(*
    private sync block removes the needs for circular interfaces variable passing amongs dependant Fbs
    that would otherwise lessen readability and complicate code scability and maintianing
    This block adds needed encapsulation for passing private data in write mode.
    it create a a communication buffer amongs synched function blocks; can also hold shareable feature implementation
    thus limititing the needs for addtional interface instantiation.
*)
{attribute 'hide_all_locals'}
FUNCTION_BLOCK FB_MotionSyncPrivate
VAR_INPUT
END_VAR
VAR_OUTPUT
END_VAR
VAR
    // private vars for data exchange
    eSyncPrvAxisState : MC_AxisStates;
    bSyncPrvReset : BOOL;
    bSyncPrvEnable :BOOL;
    bSyncPrvPowerEn : BOOL;
    bSyncPrvExec : BOOL;
    bSyncPrvError : BOOL;
    nSyncPrvErrorID : UDINT;
    bSyncPrvHomeBusy : BOOL;
    bSyncPrvLimHit : BOOL ;
    bSyncPrvMoveBusy : BOOL;
    bSyncPrvMoveDone : BOOL;
    bSyncPrvNewMoveReq : BOOL;
    bSyncPrvAllFwdEn: BOOL:=FALSE;
    bSyncPrvAllBwdEn: BOOL:=FALSE;
    bSyncPrvAllEn: BOOL:=FALSE;
    bSyncPrvLimFwd : BOOL:=FALSE;
    bSyncPrvLimBwd : BOOL:=FALSE;
    bSyncPrvHome: BOOL:=TRUE;
    bSyncPrvRestoreDone 	: BOOL;
    bSyncPrvExecHome : BOOL;
    bSyncPrvExecMove : BOOL;
    bSyncPrvStart    : BOOL;
    bSyncPrvInterlockOk : BOOL;
    bSyncPrvAxisError	: BOOL;
    bSyncPrvAbortDone : BOOL;
    bSyncPrvCmdExecute : BOOL;
    bSyncPrvStandStill : BOOL;
    sSyncPrvErrorMessage : STRING;
    eSyncPrvMoveMode : E_EpicsMotorCmd := E_EpicsMotorCmd.MOVE_ABSOLUTE;
END_VAR

(*
    Check all post condition before updating bCommandedMoveAbsolute
    The implmentatation will depend on the axis type
    DS402 NC/Direct axis : Implementation need to check that the drive is in the correct mode before initaiting the move then set bCommandedMoveAbsolute
    MP NC axis : will immediately write to bCommandedMoveAbsolute
*)
METHOD StartMove : BOOL
VAR_INPUT
END_VAR
// Notified sync FB that a new move request is to be processed
// the receiving MotionAxis must reset this bit after getting the notification
bSyncPrvStart := TRUE;
StartMove := bSyncPrvStart ;
END_METHOD

PROPERTY INTERNAL SyncPrvAbortDone : Bool
GET
SyncPrvAbortDone := bSyncPrvAbortDone;
END_GET
SET
bSyncPrvAbortDone := SyncPrvAbortDone;
END_SET
END_PROPERTY

PROPERTY INTERNAL SyncPrvAllBwdEn : BOOL
GET
SyncPrvAllBwdEn := bSyncPrvAllBwdEn;
END_GET
SET
bSyncPrvAllBwdEn := SyncPrvAllBwdEn;
END_SET
END_PROPERTY

PROPERTY INTERNAL SyncPrvAllEn : BOOL
GET
SyncPrvAllEn := bSyncPrvAllEn;
END_GET
SET
bSyncPrvAllEn := SyncPrvAllEn;
END_SET
END_PROPERTY

PROPERTY INTERNAL SyncPrvAllFwdEn : BOOL
GET
SyncPrvAllFwdEn := bSyncPrvAllFwdEn;
END_GET
SET
bSyncPrvAllFwdEn := SyncPrvAllFwdEn;
END_SET
END_PROPERTY

PROPERTY SyncPrvAxisError : BOOL
GET
SyncPrvAxisError := bSyncPrvAxisError;
END_GET
SET
bSyncPrvAxisError := SyncPrvAxisError;
END_SET
END_PROPERTY

METHOD INTERNAL SyncPrvAxisShareRead : BOOL
// add more as needed
VAR_INPUT
    AxisState : MC_AxisStates;
    MoveBusy : BOOL;
    HomeBusy : BOOL;
    MoveDone : BOOL;
    AbortDone : BOOL;
END_VAR
END_METHOD

METHOD INTERNAL SyncPrvAxisShareWrite
// add more as needed
VAR_INPUT
    AxisState : MC_AxisStates;
    MoveBusy : BOOL;
    HomeBusy : BOOL;
    MoveDone : BOOL;
    AbortDone : BOOL;
END_VAR
END_METHOD

PROPERTY INTERNAL SyncPrvAxisState : MC_AxisStates
GET
SyncPrvAxisState := eSyncPrvAxisState;
END_GET
SET
eSyncPrvAxisState := SyncPrvAxisState;
END_SET
END_PROPERTY

PROPERTY INTERNAl SyncPrvCmdExecute : Bool
GET
SyncPrvCmdExecute := bSyncPrvCmdExecute;
END_GET
SET
bSyncPrvCmdExecute := SyncPrvCmdExecute;
END_SET
END_PROPERTY

PROPERTY INTERNAL SyncPrvEnable : BOOL
GET
SyncPrvEnable := bSyncPrvEnable;
END_GET
SET
bSyncPrvEnable := SyncPrvEnable;
END_SET
END_PROPERTY

PROPERTY INTERNAL SyncPrvError : BOOL
GET
SyncPrvError := bSyncPrvError;
END_GET
SET
bSyncPrvError := SyncPrvError;
END_SET
END_PROPERTY

PROPERTY INTERNAL SyncPrvErrorID : UDINT
GET
SyncPrvErrorID := nSyncPrvErrorID;
END_GET
SET
nSyncPrvErrorID := SyncPrvErrorID;
END_SET
END_PROPERTY

PROPERTY INTERNAL SyncPrvErrorMessage : STRING
GET
SyncPrvErrorMessage := sSyncPrvErrorMessage;
END_GET
SET
sSyncPrvErrorMessage := SyncPrvErrorMessage;
END_SET
END_PROPERTY

PROPERTY INTERNAL SyncPrvExec : BOOL
GET
SyncPrvExec := bSyncPrvExec;
END_GET
SET
bSyncPrvExec := SyncPrvExec;
END_SET
END_PROPERTY

PROPERTY INTERNAL SyncPrvExecHome : BOOL
GET
SyncPrvExecHome := bSyncPrvExecHome;
END_GET
SET
bSyncPrvExecHome := SyncPrvExecHome;
END_SET
END_PROPERTY

PROPERTY INTERNAL SyncPrvExecMove : BOOL
GET
SyncPrvExecMove := bSyncPrvExecMove;
END_GET
SET
bSyncPrvExecMove := SyncPrvExecMove;
END_SET
END_PROPERTY

PROPERTY INTERNAL SyncPrvHome : BOOL
GET
SyncPrvHome := bSyncPrvHome;
END_GET
SET
bSyncPrvHome := SyncPrvHome;
END_SET
END_PROPERTY

PROPERTY INTERNAL SyncPrvHomeBusy : BOOL
GET
SyncPrvHomeBusy := bSyncPrvHomeBusy ;
END_GET
SET
bSyncPrvHomeBusy := SyncPrvHomeBusy;
END_SET
END_PROPERTY

PROPERTY SyncPrvInterlockOk : BOOL
GET
SyncPrvInterlockOk := bSyncPrvInterlockOk;
END_GET
SET
bSyncPrvInterlockOk := SyncPrvInterlockOk;
END_SET
END_PROPERTY

PROPERTY INTERNAL SyncPrvLimBwd : BOOL
GET
SyncPrvLimBwd := bSyncPrvLimBwd;
END_GET
SET
bSyncPrvLimBwd := SyncPrvLimBwd;
END_SET
END_PROPERTY

PROPERTY INTERNAL SyncPrvLimFwd : BOOL
GET
SyncPrvLimFwd := bSyncPrvLimFwd;
END_GET
SET
bSyncPrvLimFwd := SyncPrvLimFwd;
END_SET
END_PROPERTY

PROPERTY INTERNAL SyncPrvLimHit : BOOL
GET
SyncPrvLimHit := bSyncPrvLimHit;
END_GET
SET
bSyncPrvLimHit :=SyncPrvLimHit;
END_SET
END_PROPERTY

PROPERTY INTERNAL SyncPrvMoveBusy : BOOL
GET
SyncPrvMoveBusy := bSyncPrvMoveBusy;
END_GET
SET
bSyncPrvMoveBusy := SyncPrvMoveBusy;
END_SET
END_PROPERTY

PROPERTY INTERNAL SyncPrvMoveDone : BOOL
GET
SyncPrvMoveDone := bSyncPrvMoveDone;
END_GET
SET
bSyncPrvMoveDone := SyncPrvMoveDone;
END_SET
END_PROPERTY

PROPERTY SyncPrvMoveMode : E_EpicsMotorCmd
GET
SyncPrvMoveMode := eSyncPrvMoveMode;
END_GET
SET
eSyncPrvMoveMode := SyncPrvMoveMode;
END_SET
END_PROPERTY

PROPERTY INTERNAL SyncPrvNewMoveReq : BOOL
GET
SyncPrvNewMoveReq := bSyncPrvNewMoveReq;
END_GET
SET
bSyncPrvNewMoveReq := SyncPrvNewMoveReq;
END_SET
END_PROPERTY

PROPERTY INTERNAL SyncPrvPowerEn : BOOL
GET
SyncPrvPowerEn := bSyncPrvPowerEn;
END_GET
SET
bSyncPrvPowerEn := SyncPrvPowerEn;
END_SET
END_PROPERTY

PROPERTY INTERNAL SyncPrvReset : BOOL
GET
SyncPrvReset := bSyncPrvReset;
END_GET
SET
bSyncPrvReset := SyncPrvReset;
END_SET
END_PROPERTY

PROPERTY INTERNAL SyncPrvRestoreDone : BOOL
GET
SyncPrvRestoreDone := bSyncPrvRestoreDone;
END_GET
SET
bSyncPrvRestoreDone := SyncPrvRestoreDone;
END_SET
END_PROPERTY

PROPERTY INTERNAL SyncPrvStandStill : BOOL
GET
SyncPrvStandStill := bSyncPrvStandStill;
END_GET
SET
bSyncPrvStandStill := bSyncPrvStandStill;
END_SET
END_PROPERTY

PROPERTY INTERNAL SyncPrvStart : BOOL
GET
SyncPrvStart := bSyncPrvStart;
END_GET
SET
bSyncPrvStart := SyncPrvStart;
END_SET
END_PROPERTY

END_FUNCTION_BLOCK

(* stored: Version 1.1.0.1
   POU FB_MotionSyncPrivate: Id {c8657e3e-5d0e-4fad-8966-c25217ba52eb}, SpecialFunc None
   Method StartMove: Id {3d80e2c0-e431-44a4-a043-3195d6286a28}
   Property SyncPrvAbortDone: Id {6dd90901-d65a-4bbd-8bf6-8bfb90630209}
   Get Get: Id {720e183e-7c01-4607-ab7a-ae30c406a14d}
   Set Set: Id {6c245b68-f320-4630-aa5b-a75373739dd0}
   Property SyncPrvAllBwdEn: Id {f6d0f8df-5d1b-4ff4-8d72-c759807caf80}
   Get Get: Id {adc014ce-aa13-4a87-97fb-07539f9d4700}
   Set Set: Id {eea73574-3241-4bf4-8f79-f7ff5ec72934}
   Property SyncPrvAllEn: Id {c0de1886-8603-49b1-a42c-e1d3245d918a}
   Get Get: Id {af6eba22-2060-4acb-8932-1f88130efba2}
   Set Set: Id {b892ca2e-847f-43ca-a5f0-37792dea5661}
   Property SyncPrvAllFwdEn: Id {196240ef-5413-416d-b0a0-36403e6a22fd}
   Get Get: Id {eb353156-a9c5-4bf9-9328-925ec78072c1}
   Set Set: Id {715a1ed8-f189-490b-b8ae-ee360faed8ef}
   Property SyncPrvAxisError: Id {d604227f-93c9-4397-b79b-f8c609a2d1e7}
   Get Get: Id {2e4959fa-e405-4d0f-b4cd-46d19ee40b79}
   Set Set: Id {4db127ff-c579-47d6-8dcb-6bc425060b28}
   Method SyncPrvAxisShareRead: Id {f2860416-e42f-45e1-9d20-c49a4c2fcb7b}
   Method SyncPrvAxisShareWrite: Id {977956b4-a644-4c8a-896b-b6a892853915}
   Property SyncPrvAxisState: Id {60919b8b-a0ee-4b61-b888-5912d190160f}
   Get Get: Id {2a6fc420-bce2-4a3d-b8e7-0fc168de1ca2}
   Set Set: Id {78296327-b508-4ee5-b38e-cefa436e41c3}
   Property SyncPrvCmdExecute: Id {6e2d3c9f-8b42-407a-b197-5c8b3a5c4e2f}
   Get Get: Id {f7162208-73e5-46ed-802c-e15739da172a}
   Set Set: Id {741d9f12-dedd-4bb2-bea5-e4131f5313bf}
   Property SyncPrvEnable: Id {8e4e6df9-9450-4554-9644-18f90291d164}
   Get Get: Id {ea3cbcb5-5d1b-4c6a-9355-ff92c4f664cc}
   Set Set: Id {07e63cf2-67f6-4123-8b33-f12bb7df583a}
   Property SyncPrvError: Id {1b6034c0-b26d-469a-a57b-82a6b4ebb40e}
   Get Get: Id {2090a12b-697a-474d-8f07-02cf7adb2cfa}
   Set Set: Id {92c801ed-d007-4f8d-9ca0-37d8d73043c4}
   Property SyncPrvErrorID: Id {6e1d4074-3daa-45f1-a2e9-668c0069ab66}
   Get Get: Id {18206adc-d5e9-4f24-b5c5-7f277effca4f}
   Set Set: Id {d238ce9f-bdaf-46a2-a3c5-3834a8c70f01}
   Property SyncPrvErrorMessage: Id {27bea49e-d8e8-4a4f-a7e9-70cf08f0e16c}
   Get Get: Id {9dcc7512-a6f2-48db-8247-f4fec5df4b13}
   Set Set: Id {fa436d98-1c26-42f7-8c28-2a12545185c7}
   Property SyncPrvExec: Id {f59250e2-9c98-4c00-b85c-b271e1e66ae9}
   Get Get: Id {889b001c-f145-4973-a9c8-4b26c4b13927}
   Set Set: Id {415a2309-d0bb-4d9a-be5d-8503058c5b92}
   Property SyncPrvExecHome: Id {1a442731-ec14-4dff-847a-8a074dcfe1ee}
   Get Get: Id {0f329710-b157-4376-ba01-676248ccb74b}
   Set Set: Id {89904ee6-5423-4c23-9689-bd4c17a9adb5}
   Property SyncPrvExecMove: Id {80544cd9-f976-4f0b-b2c4-bae73dfbe249}
   Get Get: Id {e91de8ba-593f-4ca1-8426-2d3a28014d84}
   Set Set: Id {c58577ca-2583-4536-81f7-9f68513c3f14}
   Property SyncPrvHome: Id {4a596f7b-8cd3-4101-8575-8cf898fbea0e}
   Get Get: Id {b38e456d-0618-424d-b236-77052140716c}
   Set Set: Id {af0ee15c-32ca-4568-9855-6b4fa1b56389}
   Property SyncPrvHomeBusy: Id {4dbef2a8-0478-4d7e-8785-7f84f70fd518}
   Get Get: Id {bad28b9c-c267-4ef7-af8c-55a86c0b0457}
   Set Set: Id {513660d9-a9bd-4d34-a48c-2fbb590949d5}
   Property SyncPrvInterlockOk: Id {7dbcb427-dbe7-44b9-a51b-b38b1c27ebb0}
   Get Get: Id {e01de09c-6360-4310-97b0-b651daffe994}
   Set Set: Id {b62c9b2a-1f77-4246-b9ff-95f658bd481d}
   Property SyncPrvLimBwd: Id {f32a3277-e991-4dbe-b8fd-3c81a0c59dfc}
   Get Get: Id {7473e81f-bbcc-4d89-a8c1-2765010f18e7}
   Set Set: Id {baf2e00b-623d-4734-af90-c7149b700472}
   Property SyncPrvLimFwd: Id {12a0e278-6936-49c1-85f0-c147c4f8d84a}
   Get Get: Id {754501d6-96ab-4a3f-bc61-40e52ad936a5}
   Set Set: Id {91808e78-aeef-4059-9a0d-b2a046ceed2c}
   Property SyncPrvLimHit: Id {48dba4e9-594a-4aa6-8b94-cff3ad033b6c}
   Get Get: Id {583b7193-cfed-4323-b867-2c22006efc55}
   Set Set: Id {7fed7d13-1613-4f0a-95ad-773f423ee6e8}
   Property SyncPrvMoveBusy: Id {15420f33-1dbf-440d-ad57-611e93f2e318}
   Get Get: Id {702d2cf3-0c44-4bac-b8a8-197105c16a79}
   Set Set: Id {91e71f84-421a-40b0-8aee-098563bc8eba}
   Property SyncPrvMoveDone: Id {48b7baf8-ed4e-4bb9-847e-f1327eadbca1}
   Get Get: Id {55f2c259-1d28-4c69-9ed3-51bd0af0ee15}
   Set Set: Id {96610def-86e6-4cbb-8e04-79b3050eaba1}
   Property SyncPrvMoveMode: Id {69fecb02-d639-4a28-998f-85824e41e103}
   Get Get: Id {f695e421-185b-484b-a600-ac5ab58e757f}
   Set Set: Id {ef55c95f-1908-45e9-a9cb-2b8c1f640bfa}
   Property SyncPrvNewMoveReq: Id {99d1eaeb-20b7-470e-97ca-8e71ab6dc340}
   Get Get: Id {b91286bc-c75d-4cbe-81e2-ebc4d5686439}
   Set Set: Id {dd931d0f-9513-4185-a887-4ff73f9de3a8}
   Property SyncPrvPowerEn: Id {b485bb6e-31db-4da3-a959-a64f2de8176d}
   Get Get: Id {ac508b0b-6085-4d54-ba10-918184705e91}
   Set Set: Id {273113d6-170f-4eaf-8a28-b9222afd00a2}
   Property SyncPrvReset: Id {115cac90-f6aa-4f95-a966-8d415f1cee88}
   Get Get: Id {e76d1538-b8db-4fd9-9610-382e5e0fc2f5}
   Set Set: Id {fa3aab3c-f3be-4f32-a557-a380bd9b85c0}
   Property SyncPrvRestoreDone: Id {bf833be0-1689-4371-bd70-cc4a0bf77765}
   Get Get: Id {a6680489-5f82-4020-876d-3a889009fbc1}
   Set Set: Id {72546998-d228-4251-9151-7bb114efff40}
   Property SyncPrvStandStill: Id {7184b3ef-19be-4f90-a720-16199244a90f}
   Get Get: Id {61903ec4-f58a-4936-8623-d12cf9a91c52}
   Set Set: Id {84a9c9b0-7716-4203-89dd-029c0cddc13d}
   Property SyncPrvStart: Id {a10beacd-7ab3-4f95-9af4-081100f16b6b}
   Get Get: Id {f2786676-5c43-4ceb-9f7f-98fcefa36cef}
   Set Set: Id {673ce4c6-e5e2-49f3-9d75-cb3447c4e950} *)
